RoboDK station: GLUE EXAMPLE.rdk

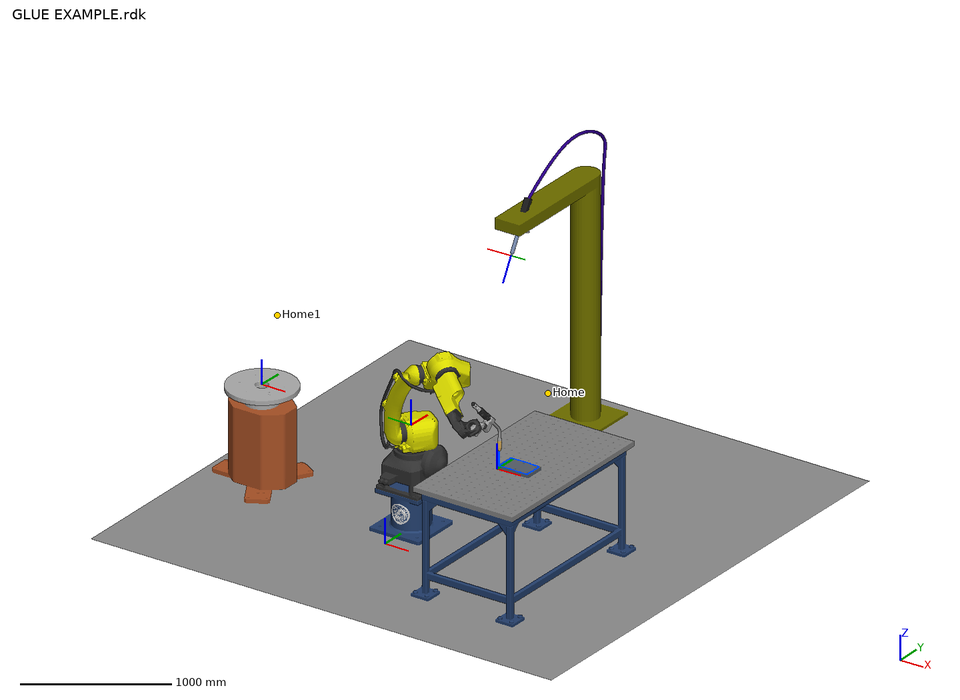
[picture v0: the station drawn from its stored meshes, robots at their saved joint values, targets as dots, program paths as lines]
Station GLUE EXAMPLE (saved by RoboDK 5.9.1). Poses are relative to the parent item; angles as X-Y-Z fixed-axis rotations.
  - frame Fanuc M-10iD/12 Base at (0, 300, 750) mm, rotated rx 0 ry 0 rz 90 deg
    - robot Fanuc M-10iD/12: 6 axes, payload 12 kg, reach 1441 mm, repeatability 0.02 mm, weight 145 kg
        modified DH rows (alpha deg, a mm, theta deg, d mm): 0, 0, 0, 450; -90, 75, -90, 0; 0, 640, 0, 0; -90, 195, 0, 700; 90, 0, 0, 0; -90, 0, 0, 75
        base shift (0, 0, -450) mm
        joint limits [-170, -90, -95, -190, -190, -450] to [170, 160, 180, 190, 190, 450]; home [-87.12, -3.54, 0.98, 0.85, -45.99, 178.78]; saved at [-124.553, 28.768, -19.522, -36.037, -98.146, 308.356]
      - tool Abicor Binzel 45deg Welding Gun, TCP at (0, 0, 400) mm, rotated rx 0 ry 45 rz 0 deg, size 179.1 x 69.8 x 552.4 mm
    - target Home1 (joint target) at (-11.12, 1067.72, 509.95) mm, rotated rx 180 ry 0 rz -90 deg; joints [90.871, -3.548, 0.989, 0.856, -45.995, 178.79] of Fanuc M-10iD/12
    - target Home (joint target) at (48.59, -1066.77, 509.83) mm, rotated rx 179.99 ry 0 rz 92 deg; joints [-87.12, -3.54, 0.98, 0.85, -45.99, 178.78] of Fanuc M-10iD/12
    - target Home (joint target) at (48.59, -1066.77, 509.83) mm, rotated rx 179.99 ry 0 rz 92 deg; joints [-87.12, -3.54, 0.98, 0.85, -45.99, 178.78] of Fanuc M-10iD/12
    - target Home (joint target) at (48.59, -1066.77, 509.83) mm, rotated rx 179.99 ry 0 rz 92 deg; joints [-87.12, -3.54, 0.98, 0.85, -45.99, 178.78] of Fanuc M-10iD/12
  - frame Glue TCP at (0, 1445, 1531) mm, rotated rx -150 ry 0 rz -180 deg
  - frame KUKA KP1-V 500 Base at (-1200, 300, 710) mm
    - robot KUKA KP1-V 500: 1 axes, payload 500 kg
        modified DH rows (alpha deg, a mm, theta deg, d mm): 0, 0, 0, 0
        joint limits [-720] to [720]; home [0]; saved at [0]
    - target P1 (Cartesian target) at (172.52, 117.59, -66.56) mm; joints [0] of KUKA KP1-V 500
  - frame World at (0, 0, 0) mm
    - object Pedestal H12in (Type 1) at (0, 300, 0) mm, size 400 x 400 x 304.8 mm, geometry from Pedestal-H12in-Type-1.sld
    - object Table 1400x800x800mm at (1000, -200, 800) mm, rotated rx 0 ry 0 rz 90 deg, size 1420 x 820 x 800 mm, geometry from Table-1400x800x800mm.sld
    - object Floor at (570, 450, 0) mm, size 3000 x 3000 x 0 mm, geometry from Floor.sld
      - object Floor at (-700, 0, 0) mm, size 3000 x 3000 x 0 mm, geometry from Floor.sld
      - object Floor at (0, 650, 0) mm, size 3000 x 3000 x 0 mm, geometry from Floor.sld
        - object Floor at (-700, 0, 0) mm, size 3000 x 3000 x 0 mm, geometry from Floor.sld
    - object RoboticCell_v1 at (-390, -940, 0) mm, geometry from RoboticCell_v1.step
      - item type 7 RoboticCell_v1-21
      - item type 7 RoboticCell_v1-22
      - item type 7 RoboticCell_v1-23
      - item type 7 RoboticCell_v1-24
      - item type 7 RoboticCell_v1-28
      - item type 7 RoboticCell_v1-29
      - item type 7 RoboticCell_v1-30
      - item type 7 RoboticCell_v1-31
      - item type 7 RoboticCell_v1-32
      - item type 7 RoboticCell_v1-33
      - item type 7 RoboticCell_v1-34
      - item type 7 RoboticCell_v1-35
      - item type 7 RoboticCell_v1-36
      - item type 7 RoboticCell_v1-38
      - item type 7 RoboticCell_v1-46
      - item type 7 RoboticCell_v1-47
      - item type 7 RoboticCell_v1-48
      - item type 7 RoboticCell_v1-27
      - item type 7 RoboticCell_v1-26
      - item type 7 RoboticCell_v1-25
    - object assembly_export at (0, 2300, 0) mm, rotated rx 0 ry 0 rz -180 deg, size 400 x 1136.1 x 2122 mm, geometry from assembly_export.step
    - object Aim Robotics SD 30/55 Dispenser at (0, 1603, 1655) mm, rotated rx -150 ry 0 rz 180 deg, size 63 x 128.2 x 396.5 mm
  - frame CAD_Frame at (900, 0, 800) mm
    - object assembly_export at (0, 0, 0) mm, size 250 x 150 x 25 mm, geometry from assembly_export.step
    - object Glue_Path_Visual at (0, 0, 0) mm, geometry from er-000
  - machining project Path1 ajustes: rotZ(0) | rotX(0)*rotY(0) | rotz(0) | onStart | onPathStart | onApproach | onPoint | onRetract | onFinish | SetRPM(%1) | SetTool(%1) | Extruder(%1) | default | default | OutOnMov(%1) | OutOffMov(%1) | onPathFinish | M_RunCode(%1)
  - program Path1 (96 instructions, listed below)
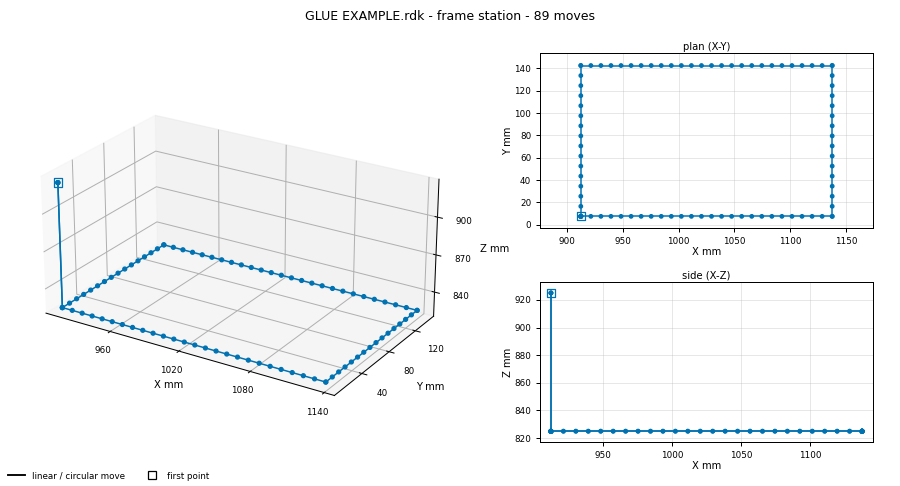
[picture p0: tool path of GLUE EXAMPLE.rdk in frame station, 89 of 89 moves have a stored position in this frame; points joined in program order, loops and branches not executed]

--- program Path1 (robot Fanuc M-10iD/12) ---
  Suave(1)
  Establecer velocidad (1000.0 mm/s)
  Est. Ref.: CAD_Frame
  Est. herr: Abicor Binzel 45deg Welding Gun
  Mostrar Abicor Binzel 45deg Welding Gun
  MoveJ 1 to (12.5, 7.5, 125) mm, rotated rx 180 ry 0 rz -90 deg; joints [-124.553, 28.768, -19.522, -36.037, -98.146, 308.356]
  MoveL 2 to (12.5, 7.5, 125) mm, rotated rx 180 ry 0 rz -90 deg; joints [-124.553, 28.768, -19.522, -36.037, -98.146, 308.356]
  MoveL 3 to (12.5, 7.5, 25) mm, rotated rx 180 ry 0 rz -90 deg; joints [-124.553, 30.052, -26.923, -35.647, -92.144, 312.705]
  MoveL 4 to (12.5, 7.5, 25) mm, rotated rx 180 ry 0 rz -90 deg; joints [-124.553, 30.052, -26.923, -35.647, -92.144, 312.705]
  Establecer velocidad (50.0 mm/s)
  MoveL 5 to (21.5, 7.5, 25) mm, rotated rx 180 ry 0 rz -90 deg; joints [-124.29, 30.743, -26.609, -35.779, -92.262, 312.332]
  MoveL 6 to (30.5, 7.5, 25) mm, rotated rx 180 ry 0 rz -90 deg; joints [-124.032, 31.44, -26.286, -35.91, -92.388, 311.954]
  MoveL 7 to (39.5, 7.5, 25) mm, rotated rx -180 ry 0 rz -90 deg; joints [-123.776, 32.146, -25.953, -36.038, -92.523, 311.573]
  MoveL 8 to (48.5, 7.5, 25) mm, rotated rx 180 ry 0 rz -90 deg; joints [-123.524, 32.859, -25.61, -36.166, -92.666, 311.187]
  MoveL 9 to (57.5, 7.5, 25) mm, rotated rx 180 ry 0 rz -90 deg; joints [-123.276, 33.581, -25.257, -36.291, -92.819, 310.796]
  MoveL 10 to (66.5, 7.5, 25) mm, rotated rx 180 ry 0 rz -90 deg; joints [-123.03, 34.312, -24.892, -36.415, -92.98, 310.401]
  MoveL 11 to (75.5, 7.5, 25) mm, rotated rx 180 ry 0 rz -90 deg; joints [-122.788, 35.052, -24.516, -36.538, -93.152, 310]
  MoveL 12 to (84.5, 7.5, 25) mm, rotated rx 180 ry 0 rz -90 deg; joints [-122.549, 35.802, -24.129, -36.659, -93.333, 309.593]
  MoveL 13 to (93.5, 7.5, 25) mm, rotated rx 180 ry 0 rz -90 deg; joints [-122.313, 36.563, -23.729, -36.78, -93.524, 309.181]
  MoveL 14 to (102.5, 7.5, 25) mm, rotated rx 180 ry 0 rz -90 deg; joints [-122.08, 37.335, -23.316, -36.899, -93.727, 308.761]
  MoveL 15 to (111.5, 7.5, 25) mm, rotated rx 180 ry 0 rz -90 deg; joints [-121.85, 38.119, -22.89, -37.018, -93.94, 308.335]
  MoveL 16 to (120.5, 7.5, 25) mm, rotated rx 180 ry 0 rz -90 deg; joints [-121.623, 38.916, -22.45, -37.136, -94.165, 307.901]
  MoveL 17 to (129.5, 7.5, 25) mm, rotated rx 180 ry 0 rz -90 deg; joints [-121.399, 39.726, -21.994, -37.254, -94.402, 307.46]
  MoveL 18 to (138.5, 7.5, 25) mm, rotated rx 180 ry 0 rz -90 deg; joints [-121.177, 40.551, -21.523, -37.371, -94.653, 307.009]
  MoveL 19 to (147.5, 7.5, 25) mm, rotated rx 180 ry 0 rz -90 deg; joints [-120.959, 41.392, -21.035, -37.489, -94.916, 306.549]
  MoveL 20 to (156.5, 7.5, 25) mm, rotated rx 180 ry 0 rz -90 deg; joints [-120.743, 42.25, -20.529, -37.607, -95.195, 306.079]
  MoveL 21 to (165.5, 7.5, 25) mm, rotated rx 180 ry 0 rz -90 deg; joints [-120.53, 43.127, -20.004, -37.726, -95.488, 305.598]
  MoveL 22 to (174.5, 7.5, 25) mm, rotated rx -180 ry 0 rz -90 deg; joints [-120.319, 44.024, -19.458, -37.845, -95.798, 305.104]
  MoveL 23 to (183.5, 7.5, 25) mm, rotated rx -180 ry 0 rz -90 deg; joints [-120.112, 44.943, -18.89, -37.966, -96.126, 304.597]
  MoveL 24 to (192.5, 7.5, 25) mm, rotated rx 180 ry 0 rz -90 deg; joints [-119.906, 45.886, -18.297, -38.089, -96.473, 304.076]
  MoveL 25 to (201.5, 7.5, 25) mm, rotated rx 180 ry 0 rz -90 deg; joints [-119.704, 46.857, -17.678, -38.214, -96.841, 303.538]
  MoveL 26 to (210.5, 7.5, 25) mm, rotated rx -180 ry 0 rz -90 deg; joints [-119.503, 47.857, -17.03, -38.342, -97.231, 302.982]
  MoveL 27 to (219.5, 7.5, 25) mm, rotated rx -180 ry 0 rz -90 deg; joints [-119.306, 48.891, -16.349, -38.473, -97.647, 302.406]
  MoveL 28 to (228.5, 7.5, 25) mm, rotated rx -180 ry 0 rz -90 deg; joints [-119.11, 49.963, -15.632, -38.609, -98.091, 301.807]
  MoveL 29 to (237.5, 7.5, 25) mm, rotated rx -180 ry 0 rz -90 deg; joints [-118.917, 51.078, -14.873, -38.75, -98.567, 301.181]
  MoveL 30 to (237.5, 7.5, 25) mm, rotated rx -180 ry 0 rz -90 deg; joints [-118.917, 51.078, -14.873, -38.75, -98.567, 301.181]
  MoveL 31 to (237.5, 16.5, 25) mm, rotated rx 180 ry 0 rz -90 deg; joints [-118.569, 50.459, -15.295, -38.841, -98.027, 301.183]
  MoveL 32 to (237.5, 25.5, 25) mm, rotated rx 180 ry 0 rz -90 deg; joints [-118.218, 49.86, -15.7, -38.936, -97.499, 301.174]
  MoveL 33 to (237.5, 34.5, 25) mm, rotated rx 180 ry 0 rz -90 deg; joints [-117.865, 49.28, -16.089, -39.035, -96.983, 301.155]
  MoveL 34 to (237.5, 43.5, 25) mm, rotated rx -180 ry 0 rz -90 deg; joints [-117.509, 48.718, -16.463, -39.138, -96.478, 301.125]
  MoveL 35 to (237.5, 52.5, 25) mm, rotated rx 180 ry 0 rz -90 deg; joints [-117.151, 48.172, -16.823, -39.245, -95.982, 301.087]
  MoveL 36 to (237.5, 61.5, 25) mm, rotated rx 180 ry 0 rz -90 deg; joints [-116.791, 47.641, -17.17, -39.355, -95.496, 301.04]
  MoveL 37 to (237.5, 70.5, 25) mm, rotated rx 180 ry 0 rz -90 deg; joints [-116.429, 47.125, -17.505, -39.468, -95.018, 300.985]
  MoveL 38 to (237.5, 79.5, 25) mm, rotated rx 180 ry 0 rz -90 deg; joints [-116.064, 46.624, -17.827, -39.583, -94.548, 300.922]
  MoveL 39 to (237.5, 88.5, 25) mm, rotated rx 180 ry 0 rz -90 deg; joints [-115.697, 46.136, -18.139, -39.702, -94.085, 300.852]
  MoveL 40 to (237.5, 97.5, 25) mm, rotated rx 180 ry 0 rz -90 deg; joints [-115.328, 45.66, -18.44, -39.823, -93.63, 300.774]
  MoveL 41 to (237.5, 106.5, 25) mm, rotated rx 180 ry 0 rz -90 deg; joints [-114.957, 45.197, -18.731, -39.946, -93.181, 300.691]
  MoveL 42 to (237.5, 115.5, 25) mm, rotated rx -180 ry 0 rz -90 deg; joints [-114.583, 44.746, -19.012, -40.072, -92.738, 300.6]
  MoveL 43 to (237.5, 124.5, 25) mm, rotated rx 180 ry 0 rz -90 deg; joints [-114.207, 44.306, -19.284, -40.2, -92.301, 300.504]
  MoveL 44 to (237.5, 133.5, 25) mm, rotated rx 180 ry 0 rz -90 deg; joints [-113.829, 43.878, -19.547, -40.329, -91.869, 300.402]
  MoveL 45 to (237.5, 142.5, 25) mm, rotated rx 180 ry 0 rz -90 deg; joints [-113.448, 43.46, -19.802, -40.46, -91.443, 300.294]
  MoveL 46 to (237.5, 142.5, 25) mm, rotated rx 180 ry 0 rz -90 deg; joints [-113.448, 43.46, -19.802, -40.46, -91.443, 300.294]
  MoveL 47 to (228.5, 142.5, 25) mm, rotated rx 180 ry 0 rz -90 deg; joints [-113.615, 42.519, -20.369, -40.392, -91.113, 300.781]
  MoveL 48 to (219.5, 142.5, 25) mm, rotated rx -180 ry 0 rz -90 deg; joints [-113.784, 41.599, -20.914, -40.325, -90.8, 301.254]
  MoveL 49 to (210.5, 142.5, 25) mm, rotated rx 180 ry 0 rz -90 deg; joints [-113.955, 40.698, -21.439, -40.258, -90.503, 301.716]
  MoveL 50 to (201.5, 142.5, 25) mm, rotated rx -180 ry 0 rz -90 deg; joints [-114.128, 39.814, -21.945, -40.191, -90.221, 302.165]
  MoveL 51 to (192.5, 142.5, 25) mm, rotated rx 180 ry 0 rz -90 deg; joints [-114.304, 38.946, -22.433, -40.124, -89.953, 302.605]
  MoveL 52 to (183.5, 142.5, 25) mm, rotated rx 180 ry 0 rz -90 deg; joints [-114.482, 38.093, -22.904, -40.056, -89.698, 303.034]
  MoveL 53 to (174.5, 142.5, 25) mm, rotated rx -180 ry 0 rz -90 deg; joints [-114.663, 37.253, -23.36, -39.988, -89.456, 303.455]
  MoveL 54 to (165.5, 142.5, 25) mm, rotated rx 180 ry 0 rz -90 deg; joints [-114.846, 36.426, -23.801, -39.92, -89.225, 303.867]
  MoveL 55 to (156.5, 142.5, 25) mm, rotated rx -180 ry 0 rz -90 deg; joints [-115.032, 35.611, -24.228, -39.85, -89.007, 304.271]
  MoveL 56 to (147.5, 142.5, 25) mm, rotated rx 180 ry 0 rz -90 deg; joints [-115.221, 34.807, -24.642, -39.78, -88.799, 304.667]
  MoveL 57 to (138.5, 142.5, 25) mm, rotated rx 180 ry 0 rz -90 deg; joints [-115.412, 34.013, -25.042, -39.709, -88.602, 305.057]
  MoveL 58 to (129.5, 142.5, 25) mm, rotated rx -180 ry 0 rz -90 deg; joints [-115.606, 33.228, -25.43, -39.636, -88.415, 305.44]
  MoveL 59 to (120.5, 142.5, 25) mm, rotated rx -180 ry 0 rz -90 deg; joints [-115.802, 32.453, -25.806, -39.562, -88.238, 305.816]
  MoveL 60 to (111.5, 142.5, 25) mm, rotated rx -180 ry 0 rz -90 deg; joints [-116.002, 31.686, -26.171, -39.486, -88.071, 306.187]
  MoveL 61 to (102.5, 142.5, 25) mm, rotated rx -180 ry 0 rz -90 deg; joints [-116.204, 30.927, -26.524, -39.409, -87.913, 306.551]
  MoveL 62 to (93.5, 142.5, 25) mm, rotated rx 180 ry 0 rz -90 deg; joints [-116.409, 30.176, -26.867, -39.331, -87.765, 306.911]
  MoveL 63 to (84.5, 142.5, 25) mm, rotated rx -180 ry 0 rz -90 deg; joints [-116.617, 29.431, -27.2, -39.25, -87.625, 307.265]
  MoveL 64 to (75.5, 142.5, 25) mm, rotated rx 180 ry 0 rz -90 deg; joints [-116.829, 28.694, -27.522, -39.168, -87.494, 307.615]
  MoveL 65 to (66.5, 142.5, 25) mm, rotated rx 180 ry 0 rz -90 deg; joints [-117.043, 27.962, -27.835, -39.084, -87.371, 307.96]
  MoveL 66 to (57.5, 142.5, 25) mm, rotated rx 180 ry 0 rz -90 deg; joints [-117.261, 27.237, -28.138, -38.998, -87.257, 308.301]
  MoveL 67 to (48.5, 142.5, 25) mm, rotated rx 180 ry 0 rz -90 deg; joints [-117.482, 26.517, -28.432, -38.909, -87.15, 308.637]
  MoveL 68 to (39.5, 142.5, 25) mm, rotated rx 180 ry 0 rz -90 deg; joints [-117.706, 25.802, -28.717, -38.819, -87.052, 308.969]
  MoveL 69 to (30.5, 142.5, 25) mm, rotated rx 180 ry 0 rz -90 deg; joints [-117.934, 25.093, -28.992, -38.726, -86.962, 309.298]
  MoveL 70 to (21.5, 142.5, 25) mm, rotated rx 180 ry 0 rz -90 deg; joints [-118.165, 24.388, -29.26, -38.631, -86.88, 309.623]
  MoveL 71 to (12.5, 142.5, 25) mm, rotated rx 180 ry 0 rz -90 deg; joints [-118.399, 23.688, -29.518, -38.534, -86.805, 309.945]
  MoveL 72 to (12.5, 142.5, 25) mm, rotated rx 180 ry 0 rz -90 deg; joints [-118.399, 23.688, -29.518, -38.534, -86.805, 309.945]
  MoveL 73 to (12.5, 133.5, 25) mm, rotated rx -180 ry 0 rz -90 deg; joints [-118.835, 24.069, -29.379, -38.331, -87.15, 310.155]
  MoveL 74 to (12.5, 124.5, 25) mm, rotated rx 180 ry 0 rz -90 deg; joints [-119.267, 24.455, -29.235, -38.129, -87.496, 310.362]
  MoveL 75 to (12.5, 115.5, 25) mm, rotated rx 180 ry 0 rz -90 deg; joints [-119.695, 24.848, -29.086, -37.929, -87.844, 310.565]
  MoveL 76 to (12.5, 106.5, 25) mm, rotated rx -180 ry 0 rz -90 deg; joints [-120.12, 25.247, -28.933, -37.73, -88.192, 310.765]
  MoveL 77 to (12.5, 97.5, 25) mm, rotated rx 180 ry 0 rz -90 deg; joints [-120.541, 25.652, -28.776, -37.532, -88.542, 310.961]
  MoveL 78 to (12.5, 88.5, 25) mm, rotated rx 180 ry 0 rz -90 deg; joints [-120.958, 26.063, -28.613, -37.336, -88.893, 311.153]
  MoveL 79 to (12.5, 79.5, 25) mm, rotated rx 180 ry 0 rz -90 deg; joints [-121.372, 26.481, -28.446, -37.141, -89.246, 311.341]
  MoveL 80 to (12.5, 70.5, 25) mm, rotated rx -180 ry 0 rz -90 deg; joints [-121.782, 26.904, -28.274, -36.948, -89.601, 311.526]
  MoveL 81 to (12.5, 61.5, 25) mm, rotated rx -180 ry 0 rz -90 deg; joints [-122.188, 27.335, -28.097, -36.757, -89.958, 311.707]
  MoveL 82 to (12.5, 52.5, 25) mm, rotated rx 180 ry 0 rz -90 deg; joints [-122.591, 27.771, -27.915, -36.568, -90.316, 311.883]
  MoveL 83 to (12.5, 43.5, 25) mm, rotated rx -180 ry 0 rz -90 deg; joints [-122.991, 28.214, -27.728, -36.38, -90.677, 312.056]
  MoveL 84 to (12.5, 34.5, 25) mm, rotated rx -180 ry 0 rz -90 deg; joints [-123.387, 28.664, -27.535, -36.194, -91.04, 312.224]
  MoveL 85 to (12.5, 25.5, 25) mm, rotated rx -180 ry 0 rz -90 deg; joints [-123.779, 29.12, -27.337, -36.009, -91.405, 312.389]
  MoveL 86 to (12.5, 16.5, 25) mm, rotated rx -180 ry 0 rz -90 deg; joints [-124.167, 29.583, -27.133, -35.827, -91.773, 312.549]
  MoveL 87 to (12.5, 7.5, 25) mm, rotated rx 180 ry 0 rz -90 deg; joints [-124.553, 30.052, -26.923, -35.647, -92.144, 312.705]
  Establecer velocidad (1000.0 mm/s)
  MoveL 88 to (12.5, 7.5, 25) mm, rotated rx 180 ry 0 rz -90 deg; joints [-124.553, 30.052, -26.923, -35.647, -92.144, 312.705]
  MoveL 89 to (12.5, 7.5, 125) mm, rotated rx 180 ry 0 rz -90 deg; joints [-124.553, 28.768, -19.522, -36.037, -98.146, 308.356]
